Fanuc KAREL source: kt00001.KL

-- PROVISIONAL review KL for V770-1; original PC SHA256 ac1aa06de9db6b206a4049c6fa9c26d68c2c329281e4460f54376bf1525b35b4
-- Incomplete behavior may be omitted. Consult companion uncertainty JSON. Do not deploy.
PROGRAM KT00001
%NOLOCKGROUP
VAR
  I1 : INTEGER
  I2 : INTEGER
  OUT : INTEGER
BEGIN
  -- UNRESOLVED_PC offsets 5-16; opcodes 2E,23
  -- UNRESOLVED_PC offsets 21-32; opcodes 2E,23
  -- UNRESOLVED_PC offsets 37-48; opcodes 2E,23
  -- UNRESOLVED_PC offsets 53-64; opcodes 2E,23
  -- UNRESOLVED_PC offsets 69-88; opcodes 21,21,52,23
  -- UNRESOLVED_PC offsets 93-97; opcodes 7F
END KT00001
